// SIMATIC STEP 7 (V5.x) project PLC_NAKAT
// CPU: CPU 315-2 PN/DP
// station: Hardware
// station: VIPA
// station: P_ADR_BUS
// program: S7 Program(1)

SYMBOL_TABLE
"TO_PRV"	DB 200	DB 200
"FROM_PRV"	DB 201	DB 201
"oscilaciya"	FB 1	FB 1
"AI_dat"	FB 2	FB 2
"GKS_Hydrostation"	FB 3	FB 3
"regul_privod"	FB 4	FB 4
"pryzhym_tVala_mode"	FB 5	FB 5
"SCALE"	FC 104	FC 104	// Scaling Values
"Read Analog Value 464-2"	FC 105	FC 105	// Read Analog Value 464-2
"UNSCALE"	FC 106	FC 106	// Unscaling Values
"x0"	I 0.0	BOOL	// реле температури
"x4"	I 0.1	BOOL	// реле тиску S6 вилка
"x1"	I 0.2	BOOL	// Рівень масла
"x5"	I 0.3	BOOL	// реле тиску S7 тамбурний вал
"x6"	I 0.5	BOOL	// фільтр S1 каландр
"x3"	I 0.6	BOOL	// реле тиску S5 каландр
"x7"	I 0.7	BOOL	// фільтр S2 вилка
"x8"	I 1.0	BOOL	// фільтр S3 тамбурний вал
"x37"	I 4.3	BOOL	// осциляція ручний старт
"x39"	I 4.7	BOOL	// осциляція авто
"x64"	I 8.0	BOOL	// переключатель замки поворотного рычага вилка nc
"x68"	I 8.1	BOOL	// переключатель прижим тамбурного вала свести
"x65"	I 8.2	BOOL	// переключатель замки поворотного рычага вилка no
"x69"	I 8.3	BOOL	// переключатель прижим тамбурного вала отвести
"x66"	I 8.4	BOOL	// переключатель вилка поднять
"x70"	I 8.5	BOOL	// перемикач перезаправка наката Р/А
"x67"	I 8.6	BOOL	// переключатель вилка опустить
"x71"	I 8.7	BOOL	// перемикач тормоз тамбура
"x72"	I 9.0	BOOL	// каландр насос А вибір
"x80"	I 9.1	BOOL	// гідронасос А (вилка) вибір
"x73"	I 9.2	BOOL	// каландр насос В вибір
"x81"	I 9.3	BOOL	// гідронасос В (вилка) вибір
"x76"	I 9.4	BOOL	// кюстерс насос А вибір
"x84"	I 9.5	BOOL	// гидронасос А прижима тамбурного вала выбор
"x77"	I 9.6	BOOL	// кюстерс насос В вибір
"x85"	I 9.7	BOOL	// гидронасос В прижима тамбурного вала выбор
"x101"	I 11.3	BOOL	// ключ безпеки накат
"x102"	I 11.5	BOOL	// ключ робота
"x108"	I 12.1	BOOL	// кнопка накат подтянуть
"x109"	I 12.3	BOOL	// ключ безпеки розгонний тамбур
"x106"	I 12.4	BOOL	// кнопка накат стоп
"x110"	I 12.5	BOOL	// розгонний тамбур стоп
"x107"	I 12.6	BOOL	// кнопка пуск накат
"x111"	I 12.7	BOOL	// розгонний тамбур пуск
"x135"	I 15.7	BOOL	// Замки
"x136"	I 16.0	BOOL	// Вилка в нижньому положенні
"x137"	I 16.2	BOOL	// прижимний вал в режимі дозволу
"x74"	I 17.0	BOOL	// каландр насос А старт
"x82"	I 17.1	BOOL	// гідронасос А (вилка) старт
"x75"	I 17.2	BOOL	// каландр насос В старт
"x83"	I 17.3	BOOL	// гідронасос В (вилка) старт
"x78"	I 17.4	BOOL	// кюстерс насос А старт
"x86"	I 17.5	BOOL	// гидронасос А прижима тамбурного вала старт
"x79"	I 17.6	BOOL	// кюстерс насос В старт
"x87"	I 17.7	BOOL	// гидронасос В прижима тамбурного вала старт
"GKS_ready"	M 10.0	BOOL	// готовність GKS
"gks_alm"	M 10.2	BOOL	// відсутність готовності
"osc_nakat"	M 10.3	BOOL
"nakat_on"	M 200.0	BOOL
"rTambur_on"	M 200.2	BOOL
"kvit"	M 1000.0	BOOL	// квитирование аварии
"PI3"	PIW 272	INT
"PI5"	PIW 274	INT
"PI4"	PIW 276	INT
"PI6"	PIW 278	INT
"Y2_FS"	PIW 280	INT
"temp2"	PIW 282	INT
"Y2_TS"	PIW 284	INT
"temp4"	PIW 286	INT
"AI3_1"	PIW 288	INT
"AI3_2"	PIW 290	INT
"AI3_3"	PIW 292	INT
"AI3_4"	PIW 294	INT
"Y3_Stanina"	PIW 296	INT
"y2"	Q 1.1	BOOL	// прижим тамбурного вала СВЕСТИ
"y14"	Q 1.2	BOOL	// вилка поднять
"y3"	Q 1.3	BOOL	// прижим тамбурного вала ОТВЕСТИ
"y15"	Q 1.4	BOOL	// вилка опустить
"Y1_1"	Q 1.5	BOOL
"Y1"	Q 1.6	BOOL
"out23"	Q 4.3	BOOL	// гидронасос В прижима тамбурного вала
"out24"	Q 4.5	BOOL	// гидронасос А прижима тамбурного вала
"out25"	Q 4.7	BOOL	// гідронасос В (вилка)
"out26"	Q 5.0	BOOL	// гідронасос А (вилка)
"out30"	Q 5.1	BOOL	// кюстерс насос В
"out27"	Q 5.2	BOOL	// каландр насос В
"out31"	Q 5.3	BOOL	// захват тамбура
"out28"	Q 5.4	BOOL	// каландр насос А
"out32"	Q 5.5	BOOL	// прижим шабера
"out29"	Q 5.6	BOOL	// кюстерс насос А
"out33"	Q 5.7	BOOL	// тормоз тамбура
"out36"	Q 6.4	BOOL	// осциляція накат
"GET"	SFB 14	SFB 14	// Read Data From a Remote CPU
"gks_alm_tmr"	T 0	TIMER
"vilka_up_tmr"	T 1	TIMER
"VAT_1_RTD"	VAT 1	
"VAT_2_DI"	VAT 2	
"VAT_3_do"	VAT 3	
"VAT_4_MW"	VAT 4	
END_SYMBOL_TABLE

FUNCTION_BLOCK "oscilaciya"	// FB 1
VERSION : 0.1
BEGIN
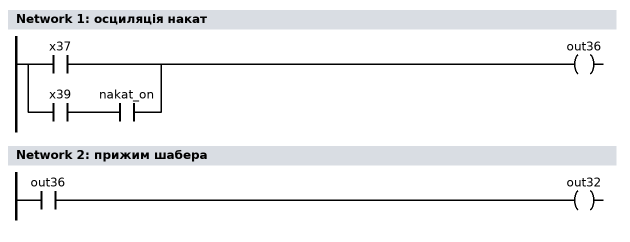
NETWORK
TITLE = осциляція накат
      O     "x37";
      O;
      A     "x39";
      A     "nakat_on";
      =     "out36";
NETWORK
TITLE = прижим шабера
      A     "out36";
      =     "out32";
END_FUNCTION_BLOCK

FUNCTION_BLOCK "AI_dat"	// FB 2
VERSION : 0.1
VAR
  PI3 : REAL ;
  PI4 : REAL ;
  PI5 : REAL ;
  PI6 : REAL ;
  Y2_FS : REAL ;
  Y2_TS : REAL ;
  Y3_stanina : REAL ;
END_VAR
VAR_TEMP
  bipolar : BOOL ;
  ret : WORD ;
  y3_stanina_int : INT ;
END_VAR
BEGIN
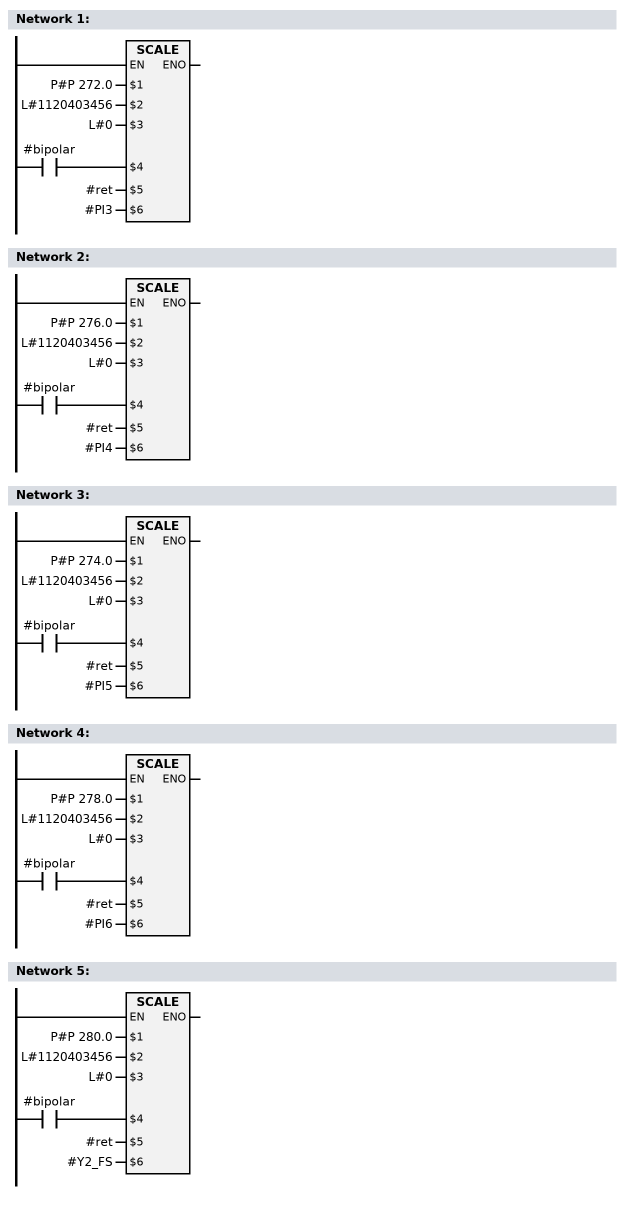
NETWORK
TITLE =
      A     #bipolar;
      =     L 6.0;
      BLD   103;
      CALL  "SCALE" (
           $1                       := P#P 272.0,
           $2                       := L#1120403456,
           $3                       := L#0,
           $4                       := L 6.0,
           $5                       := #ret,
           $6                       := #PI3);
      NOP   0;
NETWORK
TITLE =
      A     #bipolar;
      =     L 6.0;
      BLD   103;
      CALL  "SCALE" (
           $1                       := P#P 276.0,
           $2                       := L#1120403456,
           $3                       := L#0,
           $4                       := L 6.0,
           $5                       := #ret,
           $6                       := #PI4);
      NOP   0;
NETWORK
TITLE =
      A     #bipolar;
      =     L 6.0;
      BLD   103;
      CALL  "SCALE" (
           $1                       := P#P 274.0,
           $2                       := L#1120403456,
           $3                       := L#0,
           $4                       := L 6.0,
           $5                       := #ret,
           $6                       := #PI5);
      NOP   0;
NETWORK
TITLE =
      A     #bipolar;
      =     L 6.0;
      BLD   103;
      CALL  "SCALE" (
           $1                       := P#P 278.0,
           $2                       := L#1120403456,
           $3                       := L#0,
           $4                       := L 6.0,
           $5                       := #ret,
           $6                       := #PI6);
      NOP   0;
NETWORK
TITLE =
      A     #bipolar;
      =     L 6.0;
      BLD   103;
      CALL  "SCALE" (
           $1                       := P#P 280.0,
           $2                       := L#1120403456,
           $3                       := L#0,
           $4                       := L 6.0,
           $5                       := #ret,
           $6                       := #Y2_FS);
      NOP   0;
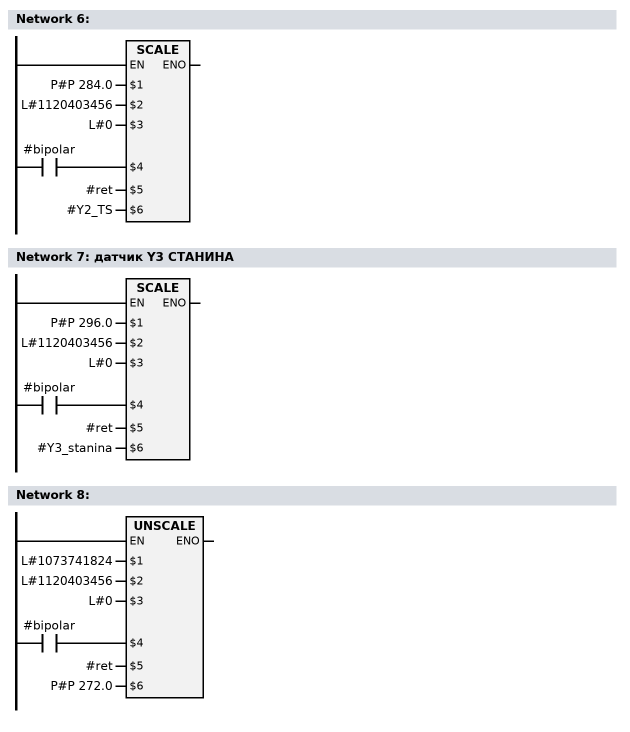
NETWORK
TITLE =
      A     #bipolar;
      =     L 6.0;
      BLD   103;
      CALL  "SCALE" (
           $1                       := P#P 284.0,
           $2                       := L#1120403456,
           $3                       := L#0,
           $4                       := L 6.0,
           $5                       := #ret,
           $6                       := #Y2_TS);
      NOP   0;
NETWORK
TITLE = датчик Y3 СТАНИНА
      A     #bipolar;
      =     L 6.0;
      BLD   103;
      CALL  "SCALE" (
           $1                       := P#P 296.0,
           $2                       := L#1120403456,
           $3                       := L#0,
           $4                       := L 6.0,
           $5                       := #ret,
           $6                       := #Y3_stanina);
      NOP   0;
NETWORK
TITLE =
      A     #bipolar;
      =     L 6.0;
      BLD   103;
      CALL  "UNSCALE" (
           $1                       := L#1073741824,
           $2                       := L#1120403456,
           $3                       := L#0,
           $4                       := L 6.0,
           $5                       := #ret,
           $6                       := P#P 272.0);
      NOP   0;
END_FUNCTION_BLOCK

FUNCTION_BLOCK "GKS_Hydrostation"	// FB 3
VERSION : 0.1
VAR_TEMP
  bypass : BOOL ;
END_VAR
BEGIN
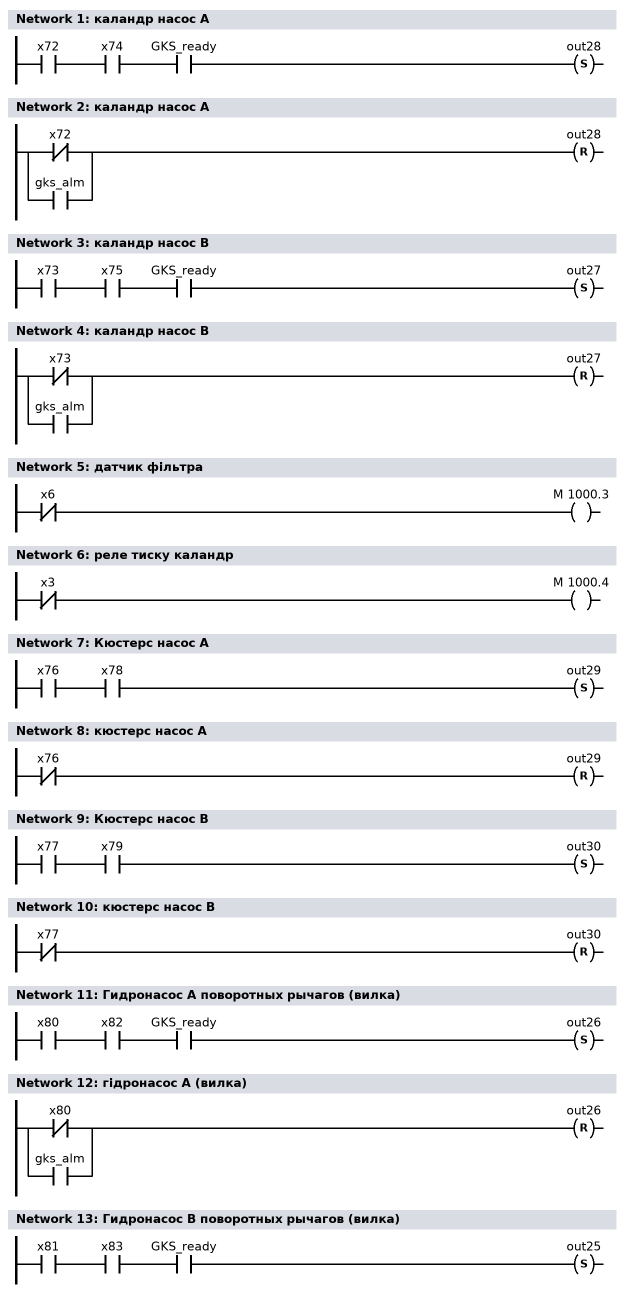
NETWORK
TITLE = каландр насос А
      A     "x72";
      A     "x74";
      A     "GKS_ready";
      S     "out28";
NETWORK
TITLE = каландр насос А
      ON    "x72";
      O     "gks_alm";
      R     "out28";
NETWORK
TITLE = каландр насос В
      A     "x73";
      A     "x75";
      A     "GKS_ready";
      S     "out27";
NETWORK
TITLE = каландр насос В
      ON    "x73";
      O     "gks_alm";
      R     "out27";
NETWORK
TITLE = датчик фільтра
      AN    "x6";
      =     M 1000.3;
NETWORK
TITLE = реле тиску каландр
      AN    "x3";
      =     M 1000.4;
NETWORK
TITLE = Кюстерс насос А 
      A     "x76";
      A     "x78";
      S     "out29";
NETWORK
TITLE = кюстерс насос А
      AN    "x76";
      R     "out29";
NETWORK
TITLE = Кюстерс насос B 
      A     "x77";
      A     "x79";
      S     "out30";
NETWORK
TITLE = кюстерс насос В
      AN    "x77";
      R     "out30";
NETWORK
TITLE = Гидронасос А поворотных рычагов (вилка)
      A     "x80";
      A     "x82";
      A     "GKS_ready";
      S     "out26";
NETWORK
TITLE = гідронасос А (вилка)
      ON    "x80";
      O     "gks_alm";
      R     "out26";
NETWORK
TITLE = Гидронасос B поворотных рычагов (вилка)
      A     "x81";
      A     "x83";
      A     "GKS_ready";
      S     "out25";
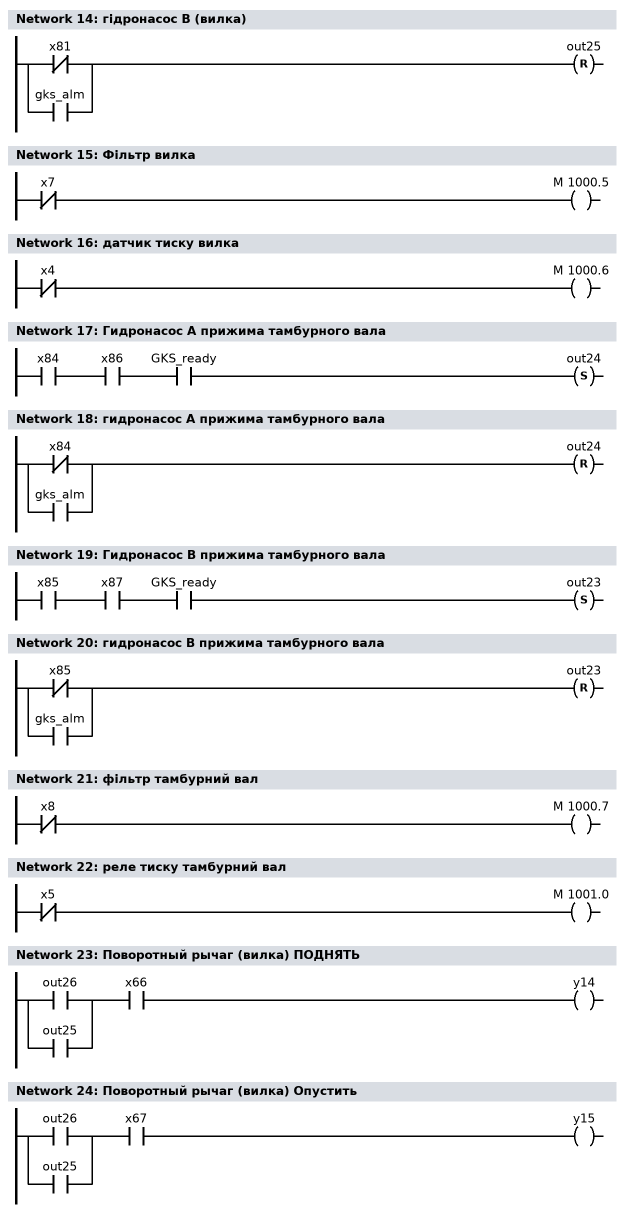
NETWORK
TITLE = гідронасос В (вилка)
      ON    "x81";
      O     "gks_alm";
      R     "out25";
NETWORK
TITLE = Фільтр вилка
      AN    "x7";
      =     M 1000.5;
NETWORK
TITLE = датчик тиску вилка
      AN    "x4";
      =     M 1000.6;
NETWORK
TITLE = Гидронасос A прижима тамбурного вала
      A     "x84";
      A     "x86";
      A     "GKS_ready";
      S     "out24";
NETWORK
TITLE = гидронасос А прижима тамбурного вала
      ON    "x84";
      O     "gks_alm";
      R     "out24";
NETWORK
TITLE = Гидронасос B прижима тамбурного вала
      A     "x85";
      A     "x87";
      A     "GKS_ready";
      S     "out23";
NETWORK
TITLE = гидронасос В прижима тамбурного вала
      ON    "x85";
      O     "gks_alm";
      R     "out23";
NETWORK
TITLE = фільтр тамбурний вал
      AN    "x8";
      =     M 1000.7;
NETWORK
TITLE = реле тиску тамбурний вал
      AN    "x5";
      =     M 1001.0;
NETWORK
TITLE = Поворотный рычаг (вилка) ПОДНЯТЬ
      A(;
      O     "out26";
      O     "out25";
      );
      A     "x66";
      =     "y14";
NETWORK
TITLE = Поворотный рычаг (вилка) Опустить
      A(;
      O     "out26";
      O     "out25";
      );
      A     "x67";
      =     "y15";
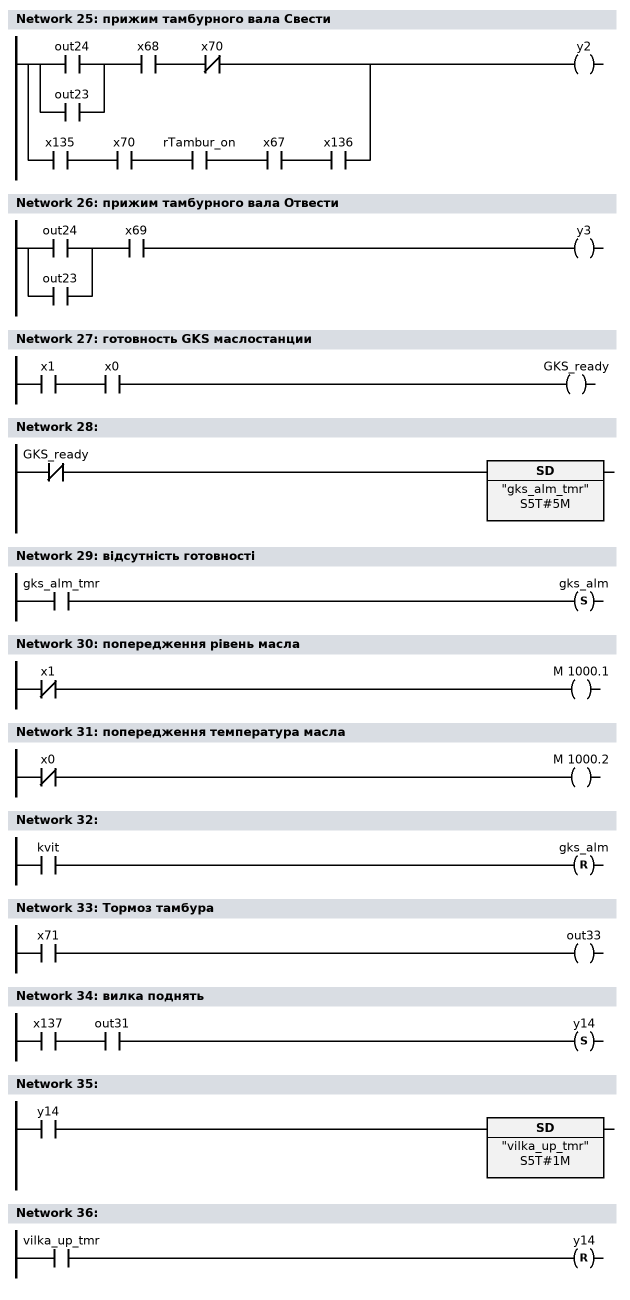
NETWORK
TITLE = прижим тамбурного вала Свести
      A(;
      O     "out24";
      O     "out23";
      );
      A     "x68";
      AN    "x70";
      O;
      A     "x135";
      A     "x70";
      A     "rTambur_on";
      A     "x67";
      A     "x136";
      =     "y2";
NETWORK
TITLE = прижим тамбурного вала Отвести
      A(;
      O     "out24";
      O     "out23";
      );
      A     "x69";
      =     "y3";
NETWORK
TITLE = готовность GKS маслостанции
      A     "x1";
      A     "x0";
      =     "GKS_ready";
NETWORK
TITLE =
      AN    "GKS_ready";
      L     S5T#5M;
      SD    "gks_alm_tmr";
NETWORK
TITLE = відсутність готовності
      A     "gks_alm_tmr";
      S     "gks_alm";
NETWORK
TITLE = попередження рівень масла
      AN    "x1";
      =     M 1000.1;
NETWORK
TITLE = попередження температура масла
      AN    "x0";
      =     M 1000.2;
NETWORK
TITLE =
      A     "kvit";
      R     "gks_alm";
NETWORK
TITLE = Тормоз тамбура
      A     "x71";
      =     "out33";
NETWORK
TITLE = вилка поднять
      A     "x137";
      A     "out31";
      S     "y14";
NETWORK
TITLE =
      A     "y14";
      L     S5T#1M;
      SD    "vilka_up_tmr";
NETWORK
TITLE =
      A     "vilka_up_tmr";
      R     "y14";
NETWORK
TITLE = робота в режимі регулювання прижиму тамбурного вала
//*******************************************************************************
END_FUNCTION_BLOCK

FUNCTION_BLOCK "regul_privod"	// FB 4
VERSION : 0.1
VAR_TEMP
  bypass : BOOL ;
END_VAR
BEGIN
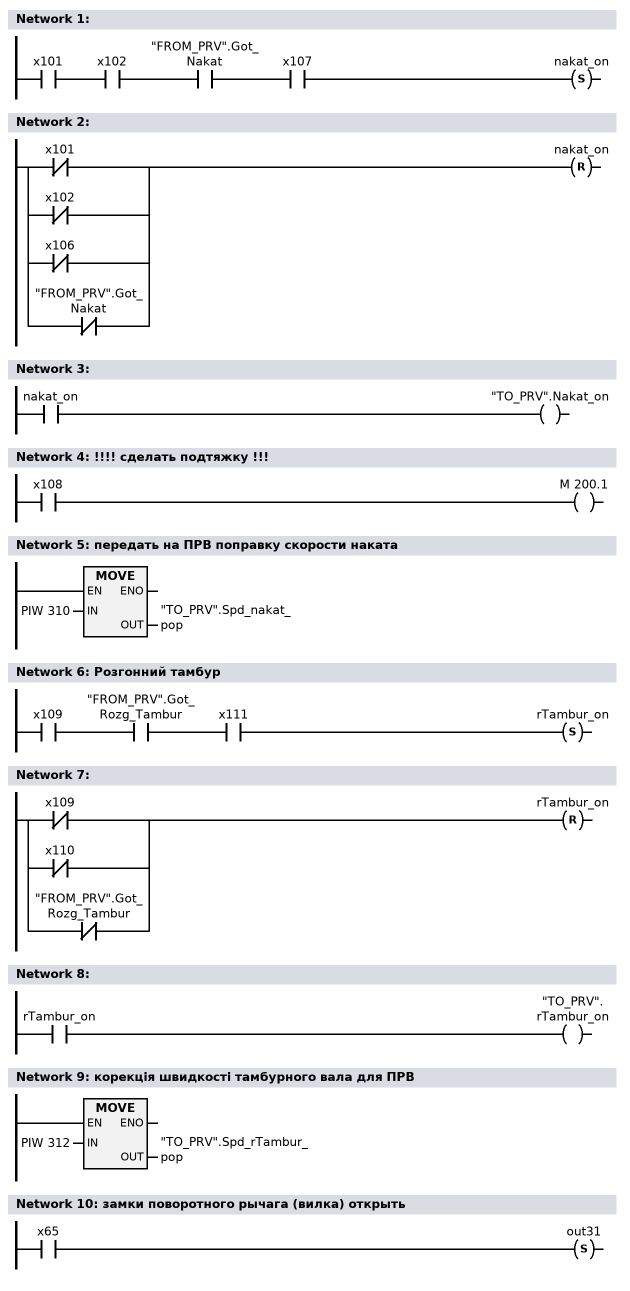
NETWORK
TITLE =
      A     "x101";
      A     "x102";
      A     "FROM_PRV".Got_Nakat;
      A     "x107";
      S     "nakat_on";
NETWORK
TITLE =
      ON    "x101";
      ON    "x102";
      ON    "x106";
      ON    "FROM_PRV".Got_Nakat;
      R     "nakat_on";
NETWORK
TITLE =
      A     "nakat_on";
      =     "TO_PRV".Nakat_on;
NETWORK
TITLE = !!!! сделать подтяжку !!!
      A     "x108";
      =     M 200.1;
NETWORK
TITLE = передать на ПРВ поправку скорости наката
      L     PIW 310;
      T     "TO_PRV".Spd_nakat_pop;
      NOP   0;
NETWORK
TITLE = Розгонний тамбур
      A     "x109";
      A     "FROM_PRV".Got_Rozg_Tambur;
      A     "x111";
      S     "rTambur_on";
NETWORK
TITLE =
      ON    "x109";
      ON    "x110";
      ON    "FROM_PRV".Got_Rozg_Tambur;
      R     "rTambur_on";
NETWORK
TITLE =
      A     "rTambur_on";
      =     "TO_PRV".rTambur_on;
NETWORK
TITLE = корекція швидкості тамбурного вала для ПРВ
      L     PIW 312;
      T     "TO_PRV".Spd_rTambur_pop;
      NOP   0;
NETWORK
TITLE = замки поворотного рычага (вилка) открыть
      A     "x65";
      S     "out31";
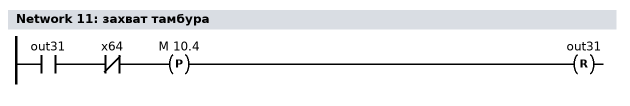
NETWORK
TITLE = захват тамбура
      A     "out31";
      AN    "x64";
      FP    M 10.4;
      R     "out31";
END_FUNCTION_BLOCK

FUNCTION_BLOCK "pryzhym_tVala_mode"	// FB 5
//Робота в режимі прижиму тамбурного вала
VERSION : 0.1
BEGIN
NETWORK
TITLE =
END_FUNCTION_BLOCK

// FC 104: know-how protected block, not included

// FC 106: know-how protected block, not included

DATA_BLOCK DB 1
VERSION : 0.0
"oscilaciya"
BEGIN
END_DATA_BLOCK

DATA_BLOCK DB 2
VERSION : 0.0
"AI_dat"
BEGIN
END_DATA_BLOCK

DATA_BLOCK DB 3
VERSION : 0.0
"GKS_Hydrostation"
BEGIN
END_DATA_BLOCK

DATA_BLOCK DB 4
VERSION : 0.0
"regul_privod"
BEGIN
END_DATA_BLOCK

DATA_BLOCK DB 14
AUTHOR : SIMATIC
FAMILY : COM_FUNC
VERSION : 0.0
"GET"
BEGIN
END_DATA_BLOCK

DATA_BLOCK "TO_PRV"	// DB 200
VERSION : 0.1
  STRUCT
   Nakat_on : BOOL ;
   rTambur_on : BOOL ;
   bool_rezerv : ARRAY  [1 .. 62 ] OF BOOL ;
   Spd_nakat_pop : INT ;
   Spd_rTambur_pop : INT ;
   int_rezerv : ARRAY  [1 .. 20 ] OF INT ;
  END_STRUCT ;	
BEGIN
END_DATA_BLOCK

DATA_BLOCK "FROM_PRV"	// DB 201
VERSION : 0.1
  STRUCT
   Got_kalandr : BOOL ;	//Gotovnist Kalandr
   Got_Rozg_Tambur : BOOL ;	//Gotovnist Rozgoni Tambur
   Got_Nakat : BOOL ;	//Gotovnist Rozgoni Nakat
   rezerv_bool : ARRAY  [1 .. 63 ] OF BOOL ;
   Speed_Suchka7_di : DINT ;
  END_STRUCT ;	
BEGIN
END_DATA_BLOCK

ORGANIZATION_BLOCK OB 1
TITLE = "Main Program Sweep (Cycle)"
VERSION : 0.1
VAR_TEMP
  OB1_EV_CLASS : BYTE ;	//Bits 0-3 = 1 (Coming event), Bits 4-7 = 1 (Event class 1)
  OB1_SCAN_1 : BYTE ;	//1 (Cold restart scan 1 of OB 1), 3 (Scan 2-n of OB 1)
  OB1_PRIORITY : BYTE ;	//Priority of OB Execution
  OB1_OB_NUMBR : BYTE ;	//1 (Organization block 1, OB1)
  OB1_RESERVED_1 : BYTE ;	//Reserved for system
  OB1_RESERVED_2 : BYTE ;	//Reserved for system
  OB1_PREV_CYCLE : INT ;	//Cycle time of previous OB1 scan (milliseconds)
  OB1_MIN_CYCLE : INT ;	//Minimum cycle time of OB1 (milliseconds)
  OB1_MAX_CYCLE : INT ;	//Maximum cycle time of OB1 (milliseconds)
  OB1_DATE_TIME : DATE_AND_TIME ;	//Date and time OB1 started
  err_GET : BOOL ;
  status_GET : WORD ;
  bypass : BOOL ;
END_VAR
BEGIN
NETWORK
TITLE = Взять данные из ПЛК_Привода
      A     M 100.3;
      =     L 25.0;
      BLD   103;
      BLD   9;
      =     L 30.0;
      CDB;
      OPN   DI 14;
      TAR2  LD 26;
      A     L 25.0;
      =     DIX 0.0;
      L     1;
      T     DIW 2;
      L     W#16#1002;
      T     DIW 8;
      L     14;
      T     DIW 10;
      L     201;
      T     DIW 12;
      L     P#DBX 0.0;
      T     DID 14;
      L     W#16#1002;
      T     DIW 48;
      L     14;
      T     DIW 50;
      L     201;
      T     DIW 52;
      L     P#DBX 0.0;
      T     DID 54;
      LAR2  P#DBX 0.0;
      UC    "GET";
      LAR2  LD 26;
      A     DIX 4.1;
      =     #err_GET;
      L     DIW 6;
      T     #status_GET;
      CDB;
      BLD   10;
      NOP   0;
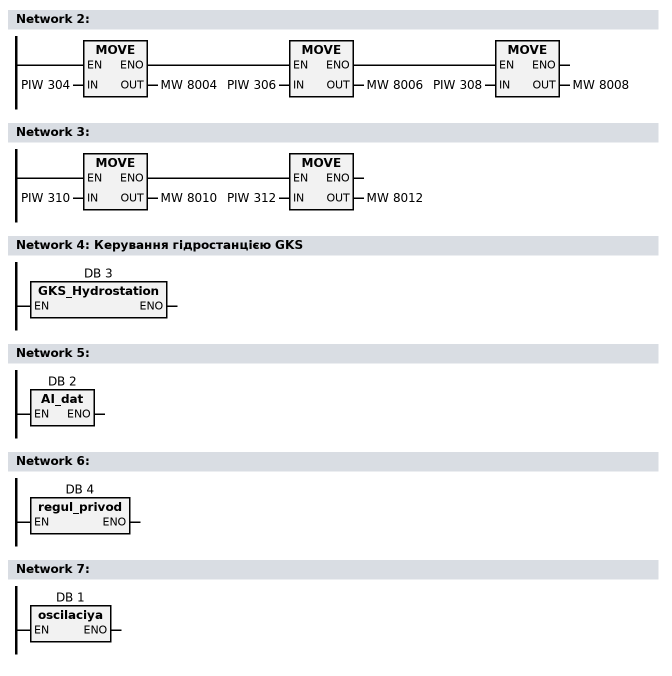
NETWORK
TITLE =
      A(;
      A(;
      L     PIW 304;
      T     MW 8004;
      SET;
      SAVE;
      CLR;
      A     BR;
      );
      JNB   _001;
      L     PIW 306;
      T     MW 8006;
      SET;
      SAVE;
      CLR;
_001: A     BR;
      );
      JNB   _002;
      L     PIW 308;
      T     MW 8008;
_002: NOP   0;
NETWORK
TITLE =
      A(;
      L     PIW 310;
      T     MW 8010;
      SET;
      SAVE;
      CLR;
      A     BR;
      );
      JNB   _003;
      L     PIW 312;
      T     MW 8012;
_003: NOP   0;
NETWORK
TITLE = Керування гідростанцією GKS
      CALL  "GKS_Hydrostation" , DB 3;
      NOP   0;
NETWORK
TITLE =
      CALL  "AI_dat" , DB 2;
      NOP   0;
NETWORK
TITLE =
      CALL  "regul_privod" , DB 4;
      NOP   0;
NETWORK
TITLE =
      CALL  "oscilaciya" , DB 1;
      NOP   0;
END_ORGANIZATION_BLOCK
